(* PLC project Tc2_Utilities.FB_LicFileRead Demo, tc3-libraries-kb TwinCAT 3.1 *)
(* stored: creationDateTime 2026-05-10T20:00:00, modificationDateTime 2026-05-10T20:00:00 *)

PROGRAM P_Demo_FB_LicFileRead
  VAR
    fbFB_LicFileRead : FB_LicFileRead;  (* Tc2_Utilities.FB_LicFileRead 实例 *)
    arg_sNetId : T_AmsNetId;  (* VAR_INPUT sNetId *)
    arg_nPort : UINT;  (* VAR_INPUT nPort *)
    arg_sFileName : STRING;  (* VAR_INPUT sFileName *)
    arg_pDestBuff : PVOID;  (* VAR_INPUT pDestBuff *)
    arg_cbReadLen : UDINT;  (* VAR_INPUT cbReadLen *)
    arg_bExecute : BOOL;  (* VAR_INPUT bExecute *)
    arg_dwPassCode : DWORD;  (* VAR_INPUT dwPassCode *)
    arg_tTimeout : TIME;  (* VAR_INPUT tTimeout *)
    out_bBusy : BOOL;  (* VAR_OUTPUT bBusy *)
    out_bError : BOOL;  (* VAR_OUTPUT bError *)
    out_nErrorId : UDINT;  (* VAR_OUTPUT nErrorId *)
    out_cbBytesread : UDINT;  (* VAR_OUTPUT cbBytesread *)
  END_VAR

            // ============================================================
// Tc2_Utilities.FB_LicFileRead 演示程序（FB 实例）
// ============================================================
// 验证步骤：
//   1. 引用 Tc2_Utilities（及依赖类型所在库 Tc2_System 等）
//   2. 编译 + 登录
//   3. 按 doc.md 给 arg_* 赋值
//   4. 在线监视 out_* / io_* 输出
// ============================================================

fbFB_LicFileRead(
    sNetId := arg_sNetId,
    nPort := arg_nPort,
    sFileName := arg_sFileName,
    pDestBuff := arg_pDestBuff,
    cbReadLen := arg_cbReadLen,
    bExecute := arg_bExecute,
    dwPassCode := arg_dwPassCode,
    tTimeout := arg_tTimeout,
    bBusy => out_bBusy,
    bError => out_bError,
    nErrorId => out_nErrorId,
    cbBytesread => out_cbBytesread
);

          
END_PROGRAM
